FUNCTION_BLOCK DOUBLE_ACTING_CYLINDER_V2 (* Basic Function Block Type *)
  (* Standard: 61499-2 *)
  (* Version 0.0, 4/29/2023, Dmitrii, Flexbridge AB, Template *)
  PACKAGE UAO.Hackathon;
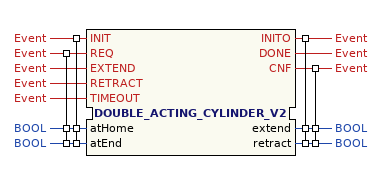
  EVENT_INPUT
    INIT WITH atEnd, atHome; (* Initialization Request *)
    REQ WITH atEnd, atHome; (* Normal Execution Request *)
    EXTEND;
    RETRACT;
    TIMEOUT;
  END_EVENT
  EVENT_OUTPUT
    INITO WITH extend, retract; (* Initialization Confirm *)
    DONE;
    CNF WITH retract, extend; (* Execution Confirmation *)
  END_EVENT
  VAR_INPUT
    atHome : BOOL; (* Input event qualifier *)
    atEnd : BOOL;
  END_VAR
  VAR_OUTPUT
    extend : BOOL; (* Output event qualifier *)
    retract : BOOL;
  END_VAR
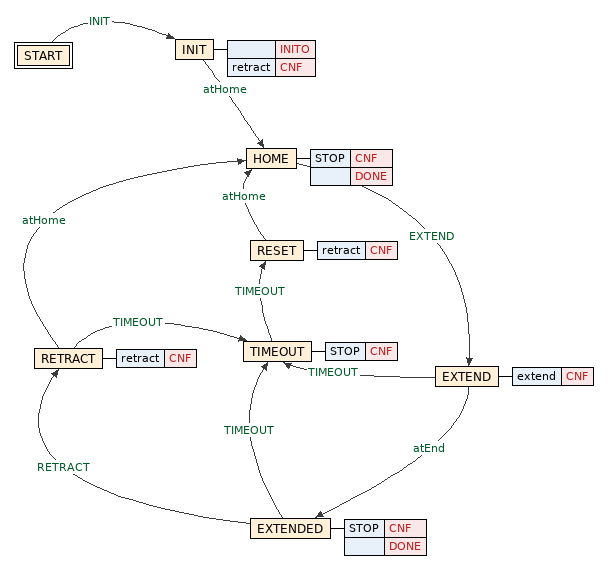
  EC_STATES
    START; (* Initial State *)
    INIT : -> INITO, retract -> CNF; (* Initialization *)
    HOME : STOP -> CNF, -> DONE;
    EXTEND : extend -> CNF;
    EXTENDED : STOP -> CNF, -> DONE;
    RETRACT : retract -> CNF;
    TIMEOUT : STOP -> CNF;
    RESET : retract -> CNF;
  END_STATES
  EC_TRANSITIONS
    START TO INIT := INIT;
    INIT TO HOME := atHome;
    HOME TO EXTEND := EXTEND;
    EXTEND TO EXTENDED := atEnd;
    EXTENDED TO RETRACT := RETRACT;
    RETRACT TO HOME := atHome;
    EXTEND TO TIMEOUT := TIMEOUT;
    RETRACT TO TIMEOUT := TIMEOUT;
    EXTENDED TO TIMEOUT := TIMEOUT;
    TIMEOUT TO RESET := TIMEOUT;
    RESET TO HOME := atHome;
  END_TRANSITIONS
  ALGORITHM INIT IN ST: (* Initialization algorithm *)
;
  END_ALGORITHM
  ALGORITHM STOP IN ST: (* Normally executed algorithm *)
extend:=FALSE;
retract:=FALSE;
  END_ALGORITHM
  ALGORITHM extend IN ST:
;
extend:=TRUE;
retract:=FALSE;
  END_ALGORITHM
  ALGORITHM retract IN ST:
;
retract:=TRUE;
extend:=FALSE;
  END_ALGORITHM
END_FUNCTION_BLOCK
